TEXTLIST P_min_indicator
  0 = 'R'
  1 = 'S'
  2 = 'T'
   = ''
END_TEXTLIST

(* stored: Version 1.1.0.1, ProductVersion 3.1.4024.11
   TextList P_min_indicator: Id {ca79d6ae-f7d5-42ce-9b9f-c6920c0cfe3b} *)
